# B&R Automation Studio project plcProject
Automation Studio 4.12.6.106

## Configuration Simulator

CPU PC_any, AutomationRuntime J4.93, Build 4.1.2, Vc V4.73.2

### Task classes (Cpu.sw)
```
Cyclic#4:
  Logic <- Logic.prg
```

### Hardware
```
PC : PC_any v1.1.1.0 (OrderNumber=PC)
  Connector IF3:
    Vnc1
    VncKeyMappingFile1 = VC\PS2-Keyboard.dis
    VncAuthentication1 = 1
    VncPasswordViewOnly1 = 0
    VncPasswordViewControl1 = 1
    VncRefreshRate1 = 100
  ConfigurationID = plcProject_Simulator
  FileDevice1
  FileDeviceName1 = USER
  FileDevicePath1 = USER_PATH
  ActivateOpcUa = 1
  OpcUaInformationModels_PV_Version = 1
```

## Logical view

### Program Logical/Logic (IEC)

#### Variables.var
```iecst
VAR
	id : STRING[80];
	cycleCounter : UDINT;
	goodProducts : UDINT;
	badProducts : UDINT;
	packMLState : STRING[80];
END_VAR
```

#### Main.st
```iecst
PROGRAM _INIT

	id := 'MACHINE_35C';
	packMLState := 'EXECUTE';

END_PROGRAM

PROGRAM _CYCLIC

	cycleCounter := cycleCounter + 1;
	goodProducts := REAL_TO_UDINT(0.9 * cycleCounter);
	badProducts := cycleCounter - goodProducts;

END_PROGRAM
```

Listed in the project but not available here: Logical/Global.typ, Logical/Global.var, Logical/Libraries
